// TIA Portal V19 export
TYPE "TExtEncoder_Sts"
// stored: Access Published
   STRUCT
      AlarmPresence : Bool;   // Cumulative alarm presence
      Standstill : Bool;   // Encoder is standstill
      InOperation : Bool;   // Encoder is in operation
      HomingDone : Bool;   // Homing done
      ActualPosition : LReal;   // Actual position
   END_STRUCT;
END_TYPE
